// TIA Portal V15.1 export
// export: Created 2024-06-21T08:41:21.4302152Z, ExportSetting WithDefaults, DisplayName Totally Integrated Automation Portal, DisplayVersion V15.1 Update 5, DisplayName TIA Portal Openness, DisplayVersion V15.1 Update 5, DisplayName SINAMICS Startdrive Advanced, DisplayVersion V15.1, DisplayName G130, G150, S120, S150, SINAMICS MV, S210, DisplayVersion V15.1, DisplayName G110M, G120, G120C, G120D, G120P, DisplayVersion V15.1, DisplayName STEP 7 Professional, DisplayVersion V15.1 Update 5, DisplayName STEP 7 Safety, DisplayVersion V15.1, DisplayName WinCC Professional, DisplayVersion V15.1 Update 5, DisplayName SIMATIC Visualization Architect, DisplayVersion V15.1
FUNCTION "LSubZoneStatus" : Void   // FC6003, FBD
TITLE = LSubzoneStatus 2017-01-24
{ S7_Optimized_Access := 'TRUE' }
VERSION : 0.1
// Convert individual subzone status bits into one UDT
// stored: AutoNumber false, IsIECCheckEnabled false, SetENOAutomatically False, UDAEnableTagReadback false
   VAR_INPUT
      I_AlarmA : Bool;   // Alarm A status of Subzone level
      I_AlarmB : Bool;   // Alarm B status of Subzone level
      I_AlarmC : Bool;   // Alarm C status of Subzone level
      I_AlarmD : Bool;   // Alarm D status of Subzone level
      I_AlarmE : Bool;   // Alarm E status (E = event) level
      I_AlarmF : Bool;   // Alarm F status of subzone level
      I_SubzoneLoaded : Bool;   // Subzone is loaded with a processed part
      I_SubZoneEmpty : Bool;   // SubZone is not loaded
      I_CycleTimeSignals : "CycleTimeSignals";   // Cycletime signals
      I_SubzoneOvercycle : Bool;   // Subzone has exceeded its' reference execution time
      I_LowRunner : Bool;   // Low runner part is present on Subzone
      I_QCheckReq : Bool;   // Quality check request
      I_QCheckOk : Bool;   // Quality check resulted in OK status
      I_QCheckNok : Bool;   // Quality check resulted in NOK status
      I_SubZoneBypass : Bool;   // Subzone in bypass
      I_BufferTooLow : Bool;   // Buffer value is below minimum level
   END_VAR
   VAR_OUTPUT
      O_SubZoneStatus : "SubzoneStatus";
   END_VAR
BEGIN

REGION Network 1: **** 1. Input **** Alarm status of the subsystem
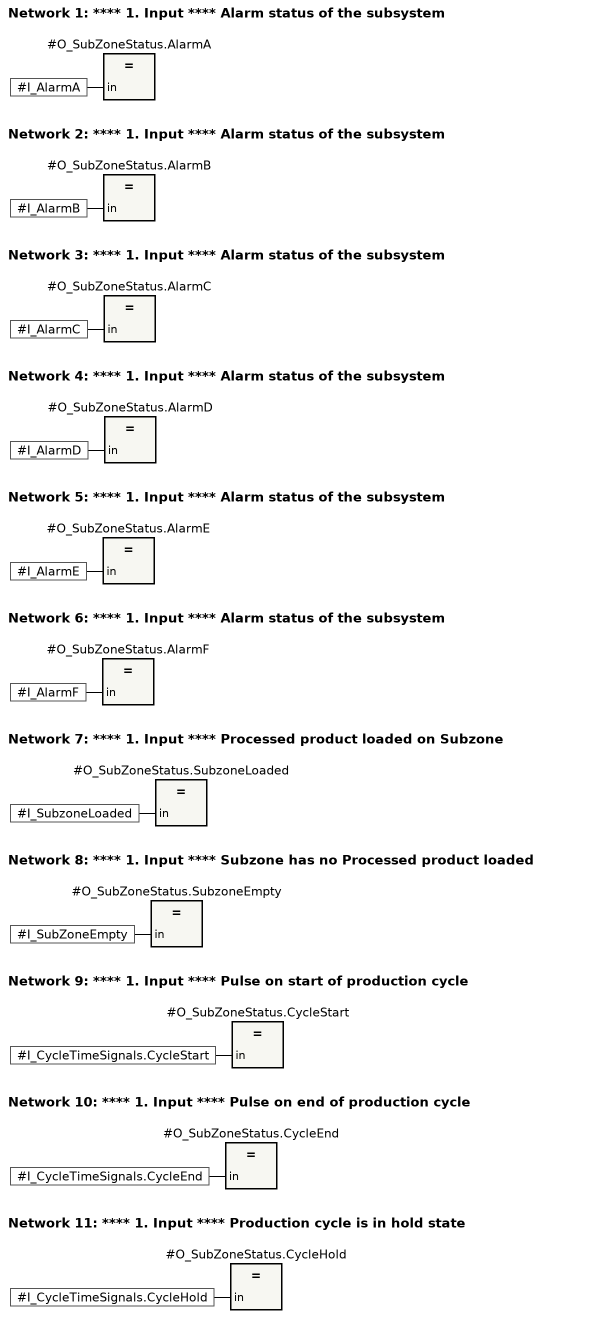
   #O_SubZoneStatus.AlarmA := #I_AlarmA;
END_REGION

REGION Network 2: **** 1. Input **** Alarm status of the subsystem
   #O_SubZoneStatus.AlarmB := #I_AlarmB;
END_REGION

REGION Network 3: **** 1. Input **** Alarm status of the subsystem
   #O_SubZoneStatus.AlarmC := #I_AlarmC;
END_REGION

REGION Network 4: **** 1. Input **** Alarm status of the subsystem
   #O_SubZoneStatus.AlarmD := #I_AlarmD;
END_REGION

REGION Network 5: **** 1. Input **** Alarm status of the subsystem
   #O_SubZoneStatus.AlarmE := #I_AlarmE;
END_REGION

REGION Network 6: **** 1. Input **** Alarm status of the subsystem
   #O_SubZoneStatus.AlarmF := #I_AlarmF;
END_REGION

REGION Network 7: **** 1. Input **** Processed product loaded on Subzone
   #O_SubZoneStatus.SubzoneLoaded := #I_SubzoneLoaded;
END_REGION

REGION Network 8: **** 1. Input **** Subzone has no Processed product loaded
   #O_SubZoneStatus.SubzoneEmpty := #I_SubZoneEmpty;
END_REGION

REGION Network 9: **** 1. Input **** Pulse on start of production cycle
   #O_SubZoneStatus.CycleStart := #I_CycleTimeSignals.CycleStart;
END_REGION

REGION Network 10: **** 1. Input **** Pulse on end of production cycle
   #O_SubZoneStatus.CycleEnd := #I_CycleTimeSignals.CycleEnd;
END_REGION

REGION Network 11: **** 1. Input **** Production cycle is in hold state
   #O_SubZoneStatus.CycleHold := #I_CycleTimeSignals.CycleHold;
END_REGION

REGION Network 12: **** 1. Input **** Infeed 1 at subzone active
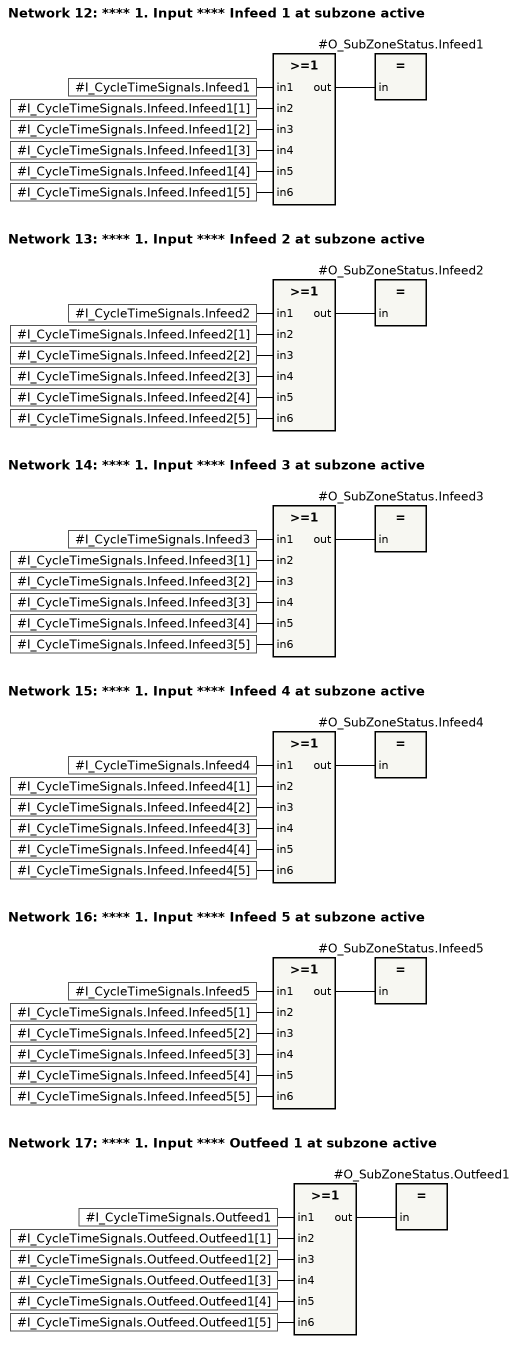
   #O_SubZoneStatus.Infeed1 := #I_CycleTimeSignals.Infeed1 OR #I_CycleTimeSignals.Infeed.Infeed1[1] OR #I_CycleTimeSignals.Infeed.Infeed1[2] OR #I_CycleTimeSignals.Infeed.Infeed1[3] OR #I_CycleTimeSignals.Infeed.Infeed1[4] OR #I_CycleTimeSignals.Infeed.Infeed1[5];
END_REGION

REGION Network 13: **** 1. Input **** Infeed 2 at subzone active
   #O_SubZoneStatus.Infeed2 := #I_CycleTimeSignals.Infeed2 OR #I_CycleTimeSignals.Infeed.Infeed2[1] OR #I_CycleTimeSignals.Infeed.Infeed2[2] OR #I_CycleTimeSignals.Infeed.Infeed2[3] OR #I_CycleTimeSignals.Infeed.Infeed2[4] OR #I_CycleTimeSignals.Infeed.Infeed2[5];
END_REGION

REGION Network 14: **** 1. Input **** Infeed 3 at subzone active
   #O_SubZoneStatus.Infeed3 := #I_CycleTimeSignals.Infeed3 OR #I_CycleTimeSignals.Infeed.Infeed3[1] OR #I_CycleTimeSignals.Infeed.Infeed3[2] OR #I_CycleTimeSignals.Infeed.Infeed3[3] OR #I_CycleTimeSignals.Infeed.Infeed3[4] OR #I_CycleTimeSignals.Infeed.Infeed3[5];
END_REGION

REGION Network 15: **** 1. Input **** Infeed 4 at subzone active
   #O_SubZoneStatus.Infeed4 := #I_CycleTimeSignals.Infeed4 OR #I_CycleTimeSignals.Infeed.Infeed4[1] OR #I_CycleTimeSignals.Infeed.Infeed4[2] OR #I_CycleTimeSignals.Infeed.Infeed4[3] OR #I_CycleTimeSignals.Infeed.Infeed4[4] OR #I_CycleTimeSignals.Infeed.Infeed4[5];
END_REGION

REGION Network 16: **** 1. Input **** Infeed 5 at subzone active
   #O_SubZoneStatus.Infeed5 := #I_CycleTimeSignals.Infeed5 OR #I_CycleTimeSignals.Infeed.Infeed5[1] OR #I_CycleTimeSignals.Infeed.Infeed5[2] OR #I_CycleTimeSignals.Infeed.Infeed5[3] OR #I_CycleTimeSignals.Infeed.Infeed5[4] OR #I_CycleTimeSignals.Infeed.Infeed5[5];
END_REGION

REGION Network 17: **** 1. Input **** Outfeed 1 at subzone active
   #O_SubZoneStatus.Outfeed1 := #I_CycleTimeSignals.Outfeed1 OR #I_CycleTimeSignals.Outfeed.Outfeed1[1] OR #I_CycleTimeSignals.Outfeed.Outfeed1[2] OR #I_CycleTimeSignals.Outfeed.Outfeed1[3] OR #I_CycleTimeSignals.Outfeed.Outfeed1[4] OR #I_CycleTimeSignals.Outfeed.Outfeed1[5];
END_REGION

REGION Network 18: **** 1. Input **** Outfeed 2 at subzone active
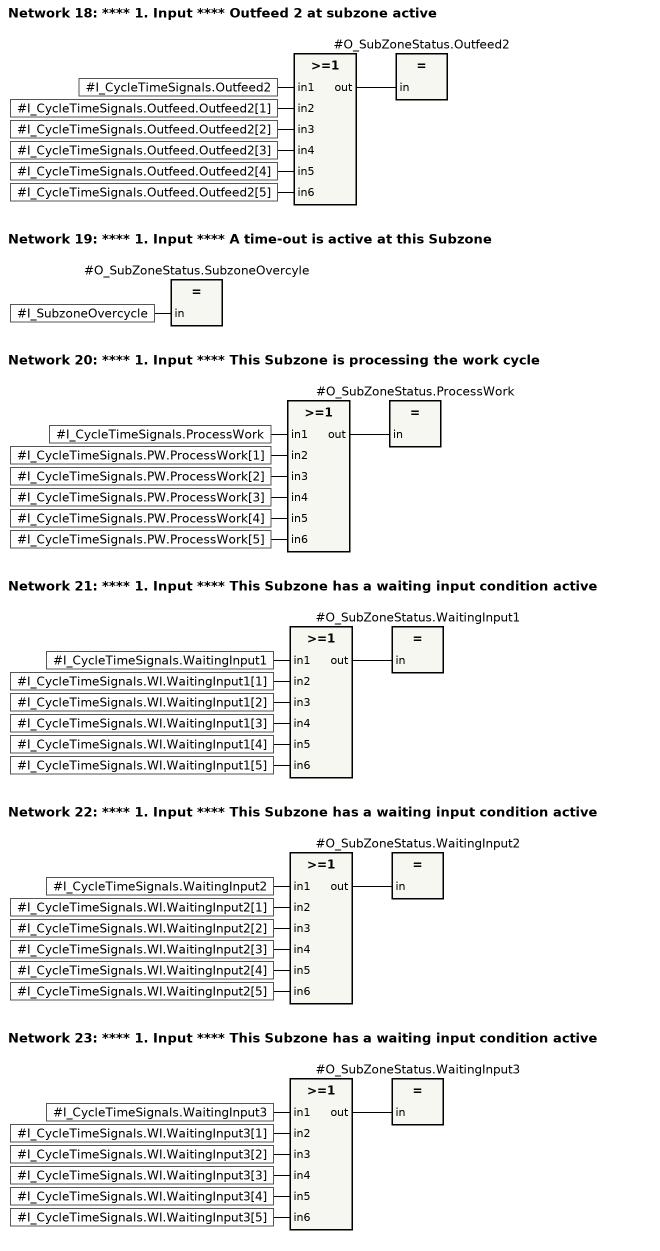
   #O_SubZoneStatus.Outfeed2 := #I_CycleTimeSignals.Outfeed2 OR #I_CycleTimeSignals.Outfeed.Outfeed2[1] OR #I_CycleTimeSignals.Outfeed.Outfeed2[2] OR #I_CycleTimeSignals.Outfeed.Outfeed2[3] OR #I_CycleTimeSignals.Outfeed.Outfeed2[4] OR #I_CycleTimeSignals.Outfeed.Outfeed2[5];
END_REGION

REGION Network 19: **** 1. Input **** A time-out is active at this Subzone
   #O_SubZoneStatus.SubzoneOvercyle := #I_SubzoneOvercycle;
END_REGION

REGION Network 20: **** 1. Input **** This Subzone is processing the work cycle
   #O_SubZoneStatus.ProcessWork := #I_CycleTimeSignals.ProcessWork OR #I_CycleTimeSignals.PW.ProcessWork[1] OR #I_CycleTimeSignals.PW.ProcessWork[2] OR #I_CycleTimeSignals.PW.ProcessWork[3] OR #I_CycleTimeSignals.PW.ProcessWork[4] OR #I_CycleTimeSignals.PW.ProcessWork[5];
END_REGION

REGION Network 21: **** 1. Input **** This Subzone has a waiting input condition active
   #O_SubZoneStatus.WaitingInput1 := #I_CycleTimeSignals.WaitingInput1 OR #I_CycleTimeSignals.WI.WaitingInput1[1] OR #I_CycleTimeSignals.WI.WaitingInput1[2] OR #I_CycleTimeSignals.WI.WaitingInput1[3] OR #I_CycleTimeSignals.WI.WaitingInput1[4] OR #I_CycleTimeSignals.WI.WaitingInput1[5];
END_REGION

REGION Network 22: **** 1. Input **** This Subzone has a waiting input condition active
   #O_SubZoneStatus.WaitingInput2 := #I_CycleTimeSignals.WaitingInput2 OR #I_CycleTimeSignals.WI.WaitingInput2[1] OR #I_CycleTimeSignals.WI.WaitingInput2[2] OR #I_CycleTimeSignals.WI.WaitingInput2[3] OR #I_CycleTimeSignals.WI.WaitingInput2[4] OR #I_CycleTimeSignals.WI.WaitingInput2[5];
END_REGION

REGION Network 23: **** 1. Input **** This Subzone has a waiting input condition active
   #O_SubZoneStatus.WaitingInput3 := #I_CycleTimeSignals.WaitingInput3 OR #I_CycleTimeSignals.WI.WaitingInput3[1] OR #I_CycleTimeSignals.WI.WaitingInput3[2] OR #I_CycleTimeSignals.WI.WaitingInput3[3] OR #I_CycleTimeSignals.WI.WaitingInput3[4] OR #I_CycleTimeSignals.WI.WaitingInput3[5];
END_REGION

REGION Network 24: **** 1. Input **** This Subzone has a waiting input condition active
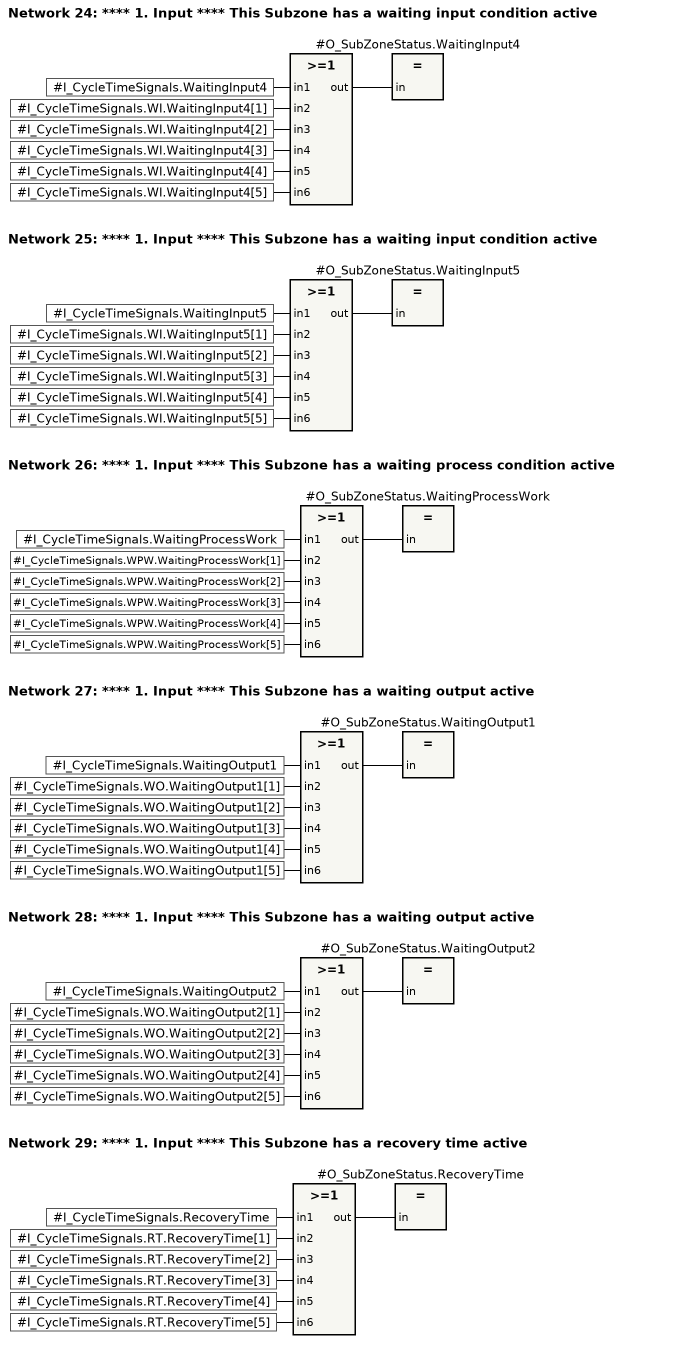
   #O_SubZoneStatus.WaitingInput4 := #I_CycleTimeSignals.WaitingInput4 OR #I_CycleTimeSignals.WI.WaitingInput4[1] OR #I_CycleTimeSignals.WI.WaitingInput4[2] OR #I_CycleTimeSignals.WI.WaitingInput4[3] OR #I_CycleTimeSignals.WI.WaitingInput4[4] OR #I_CycleTimeSignals.WI.WaitingInput4[5];
END_REGION

REGION Network 25: **** 1. Input **** This Subzone has a waiting input condition active
   #O_SubZoneStatus.WaitingInput5 := #I_CycleTimeSignals.WaitingInput5 OR #I_CycleTimeSignals.WI.WaitingInput5[1] OR #I_CycleTimeSignals.WI.WaitingInput5[2] OR #I_CycleTimeSignals.WI.WaitingInput5[3] OR #I_CycleTimeSignals.WI.WaitingInput5[4] OR #I_CycleTimeSignals.WI.WaitingInput5[5];
END_REGION

REGION Network 26: **** 1. Input **** This Subzone has a waiting process condition active
   // This Subzone has a waiting process condition active
   #O_SubZoneStatus.WaitingProcessWork := #I_CycleTimeSignals.WaitingProcessWork OR #I_CycleTimeSignals.WPW.WaitingProcessWork[1] OR #I_CycleTimeSignals.WPW.WaitingProcessWork[2] OR #I_CycleTimeSignals.WPW.WaitingProcessWork[3] OR #I_CycleTimeSignals.WPW.WaitingProcessWork[4] OR #I_CycleTimeSignals.WPW.WaitingProcessWork[5];
END_REGION

REGION Network 27: **** 1. Input **** This Subzone has a waiting output active
   #O_SubZoneStatus.WaitingOutput1 := #I_CycleTimeSignals.WaitingOutput1 OR #I_CycleTimeSignals.WO.WaitingOutput1[1] OR #I_CycleTimeSignals.WO.WaitingOutput1[2] OR #I_CycleTimeSignals.WO.WaitingOutput1[3] OR #I_CycleTimeSignals.WO.WaitingOutput1[4] OR #I_CycleTimeSignals.WO.WaitingOutput1[5];
END_REGION

REGION Network 28: **** 1. Input **** This Subzone has a waiting output active
   #O_SubZoneStatus.WaitingOutput2 := #I_CycleTimeSignals.WaitingOutput2 OR #I_CycleTimeSignals.WO.WaitingOutput2[1] OR #I_CycleTimeSignals.WO.WaitingOutput2[2] OR #I_CycleTimeSignals.WO.WaitingOutput2[3] OR #I_CycleTimeSignals.WO.WaitingOutput2[4] OR #I_CycleTimeSignals.WO.WaitingOutput2[5];
END_REGION

REGION Network 29: **** 1. Input **** This Subzone has a recovery time active
   // This Subzone has a recovery time active
   #O_SubZoneStatus.RecoveryTime := #I_CycleTimeSignals.RecoveryTime OR #I_CycleTimeSignals.RT.RecoveryTime[1] OR #I_CycleTimeSignals.RT.RecoveryTime[2] OR #I_CycleTimeSignals.RT.RecoveryTime[3] OR #I_CycleTimeSignals.RT.RecoveryTime[4] OR #I_CycleTimeSignals.RT.RecoveryTime[5];
END_REGION

REGION Network 30: **** 1. Input **** This Subzone has a lowrunner active
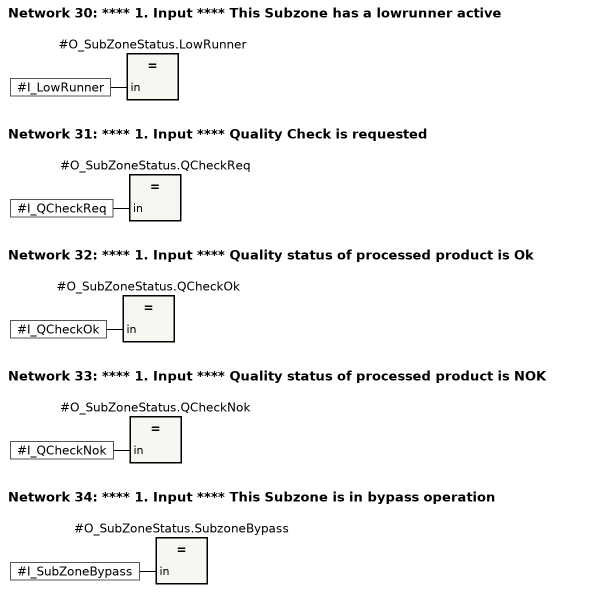
   #O_SubZoneStatus.LowRunner := #I_LowRunner;
END_REGION

REGION Network 31: **** 1. Input **** Quality Check is requested
   #O_SubZoneStatus.QCheckReq := #I_QCheckReq;
END_REGION

REGION Network 32: **** 1. Input **** Quality status of processed product is Ok
   #O_SubZoneStatus.QCheckOk := #I_QCheckOk;
END_REGION

REGION Network 33: **** 1. Input **** Quality status of processed product is NOK
   #O_SubZoneStatus.QCheckNok := #I_QCheckNok;
END_REGION

REGION Network 34: **** 1. Input **** This Subzone is in bypass operation
   #O_SubZoneStatus.SubzoneBypass := #I_SubZoneBypass;
END_REGION
END_FUNCTION
